// Mitsubishi GX Works2 project: test   PLC: Q02U

PROGRAM MAIN
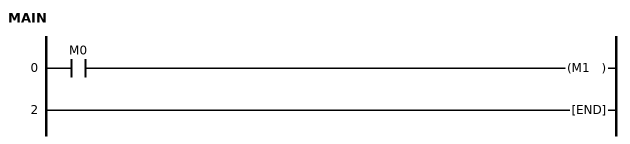
0     LD      M0
      OUT     M1
2     END
END_PROGRAM
